// TIA Portal V16 export
// export: Created 2024-12-03T15:41:40.6794035Z, ExportSetting WithDefaults, DisplayName Totally Integrated Automation Portal, DisplayVersion V16 Update 6, DisplayName TIA Portal Version Control Interface, DisplayVersion V16 Update 2, DisplayName TIA Portal Openness, DisplayVersion V16 Update 6, DisplayName TIA Portal Teamcenter Gateway, DisplayVersion V16, DisplayName SINAMICS Startdrive Advanced, DisplayVersion V16 Update 5, DisplayName SINAMICS Startdrive G130, G150, S120, S150, SINAMICS MV, S210, DisplayVersion V16 Update 5, DisplayName SINAMICS Startdrive G110M, G120, G120C, G120D, G120P, G115D, DisplayVersion V16 Update 5, DisplayName STEP 7 Professional, DisplayVersion V16 Update 6, DisplayName STEP 7 Safety, DisplayVersion V16, DisplayName WinCC Advanced / Unified PC, DisplayVersion V16 Update 6
FUNCTION_BLOCK "InstallationControl"   // FB38, SCL
{ S7_Optimized_Access := 'FALSE' }
VERSION : 0.1
// stored: AutoNumber true, IsIECCheckEnabled false, SetENOAutomatically false, UDAEnableTagReadback false
   VAR_IN_OUT
      IO_StartAutoMode : Bool;
      IO_StopAutoMode : Bool;
   END_VAR
   VAR
      zoneInstances { S7_SetPoint := 'True'} : Array[1..2] of "InstallaitonControlInstance";
   END_VAR
   VAR_TEMP
      T_Index : Int;
   END_VAR
   VAR CONSTANT
      lenght : Int := 2;
   END_VAR
BEGIN
   REGION GLOBAL STATE

       "ApplicationState_DB".GlobalState.States.AlarmActive :=
       "ApplicationState_DB".Appstate[1].Alarms.AlarmsActiveForHmi OR
       "ApplicationState_DB".Appstate[2].Alarms.AlarmsActiveForHmi OR
       "Alarms_DB".AlarmActiveShared;

       "ApplicationState_DB".GlobalState.States.EmergencyOk :=
       "ApplicationState_DB".Appstate[1].States.EmergencyOk.State OR
       "ApplicationState_DB".Appstate[2].States.EmergencyOk.State;

       "ApplicationState_DB".GlobalState.States.AutoMode :=
       "ApplicationState_DB".Appstate[1].States.AutoModeActivated.State OR
       "ApplicationState_DB".Appstate[2].States.AutoModeActivated.State;

   END_REGION

   REGION MAIN STATE

       "ApplicationState_DB".Appstate[1].States.EmergencyOk := "Inputs_DB".EMG_OK;

       "ApplicationState_DB".Appstate[1].States.ReadyForStandby := 1;
       #zoneInstances[1](IO_Appstate := "ApplicationState_DB".Appstate[1]);

       IF "Inputs_DB".Reset_System.LE THEN
           "ApplicationState_DB".Appstate[1].Hmi_Buttons.reset.SignalFromHMI := 1;
           "ApplicationState_DB".Appstate[2].Hmi_Buttons.reset.SignalFromHMI := 1;
       END_IF;



   END_REGION

   REGION STATE COPY

       FOR #T_Index := 10 TO 19 DO
           "ApplicationState_DB".Appstate[#T_Index].States := "ApplicationState_DB".Appstate[1].States;
           "ApplicationState_DB".Appstate[#T_Index].Hmi_Buttons := "ApplicationState_DB".Appstate[1].Hmi_Buttons;
       END_FOR;

       FOR #T_Index := 20 TO 29 DO
           "ApplicationState_DB".Appstate[#T_Index].States := "ApplicationState_DB".Appstate[1].States;
           "ApplicationState_DB".Appstate[#T_Index].Hmi_Buttons := "ApplicationState_DB".Appstate[1].Hmi_Buttons;
       END_FOR;

       FOR #T_Index := 30 TO 39 DO
           "ApplicationState_DB".Appstate[#T_Index].States := "ApplicationState_DB".Appstate[1].States;
           "ApplicationState_DB".Appstate[#T_Index].Hmi_Buttons := "ApplicationState_DB".Appstate[1].Hmi_Buttons;
       END_FOR;

       FOR #T_Index := 40 TO 49 DO
           "ApplicationState_DB".Appstate[#T_Index].States := "ApplicationState_DB".Appstate[1].States;
           "ApplicationState_DB".Appstate[#T_Index].Hmi_Buttons := "ApplicationState_DB".Appstate[1].Hmi_Buttons;
       END_FOR;

       FOR #T_Index := 50 TO 52 DO
           "ApplicationState_DB".Appstate[#T_Index].States := "ApplicationState_DB".Appstate[1].States;
           "ApplicationState_DB".Appstate[#T_Index].Hmi_Buttons := "ApplicationState_DB".Appstate[1].Hmi_Buttons;
       END_FOR;



   END_REGION

   REGION ALARM ACTIVE

       FOR #T_Index := 10 TO 52 DO

           "ApplicationState_DB".Appstate[#T_Index].Alarms.AlarmsActiveForHmi :=
           "ApplicationState_DB".Appstate[#T_Index].Alarms.AlarmActiveInternalPLC;

           "ApplicationState_DB".Appstate[#T_Index].Alarms.AlarmActiveInternalPLC := 0;

           IF "ApplicationState_DB".Appstate[#T_Index].Alarms.AlarmsActiveForHmi THEN
               "ApplicationState_DB".Appstate[1].Alarms.AlarmActiveInternalPLC := 1;
           END_IF;

       END_FOR;


   END_REGION

   REGION RESET CMD

       IF "HMI_DB".ResetFromHMI OR "ApplicationState_DB".Appstate[0].Hmi_Buttons.reset.SignalFromHMI THEN
           "HMI_DB".ResetFromHMI := FALSE;
           "ApplicationState_DB".Appstate[0].Hmi_Buttons.reset.SignalFromHMI := 1;
       END_IF;

   END_REGION
END_FUNCTION_BLOCK
